# B&R Automation Studio project SMA_DATA
Automation Studio 4.8.7.28 SP

## Configuration PC

CPU PC_any, AutomationRuntime M4.93, Build 6.3.0, Vc V4.73.1

### Hardware
```
PC : PC_any v1.1.1.0 (OrderNumber=PC)
  ConfigurationID = SMA_DATA_PC
  Cyclic1Duration = 10000
  Cyclic1Tolerance = 100000
  FileDevice1
  FileDeviceName1 = USER
  FileDevicePath1 = USER_PATH
  ActivateOpcUa = 1
  OpcUaInformationModels_PV_Version = 1
```

## Configuration x1586

CPU X20CP1586, AutomationRuntime J4.93, Build 6.3.0, Vc V4.73.1

### Task classes (Cpu.sw)
```
Cyclic#1:
  DataSQL <- DataSQL.prg
  DataSQLPro <- DataSQLProduct.prg
Binaries: udbdef, FWRules, TCData, iomap, ashwac, Role, sysconf, arconfig, asfw, User, ashwd
Libraries: standard, AsBrStr
```

### Hardware
```
X20CP1586 : X20CP1586 v1.13.0.0
  Connector IF1:
    ActivateIna = 0
  Connector IF2:
    ActivateDevice = 1
    Mode = Manual
    InternetAddress = 192.168.50.233
    SubnetMask = 255.255.255.0
    InaPort = 11160
    ActivateSnmp = 2
  ConfigurationID = SMA_DATA_PC
  Simulation = 1
  Cyclic1Tolerance = 100000
  FileDevice1
  FileDeviceName1 = USER
  FileDevicePath1 = USER_PATH
  ActivateOpcUa = 1
  OpcUaInformationModels_PV_Version = 1
```

## Logical view

Binary libraries used (declarations not repeated): operator, runtime, astime, AsIecCon, standard, AsBrStr

### Package Logical/Libraries - Global libraries

### GlobalDataSQL.typ
```iecst
(*Global Data SQL Struct*)

TYPE
	DataSQLOperate_typ : 	STRUCT
		RecipeRead : BOOL;
		RecipeReadStatus : UINT;
		RecipeInsert : BOOL;
		RecipeInsertReq : BOOL;
		ProductRead : BOOL;
		ProductReadStatus : UINT;
		ProductInsert : BOOL;
		ProductInsertReq : BOOL;
		AuditRead : BOOL;
		AuditReadStatus : UINT;
		AuditInsertFault : BOOL;
		AlarmRead : BOOL;
		AlarmReadStatus : UINT;
		AlarmInsertFault : BOOL;
	END_STRUCT;
END_TYPE

(*Global Data SQL Struct*)

TYPE
	DataSQLQueryConfig_typ : 	STRUCT
		StartTime : ARRAY[0..READ_QUERY_SIZE_MINUS]OF STRING[20];
		EndTime : ARRAY[0..READ_QUERY_SIZE_MINUS]OF STRING[20];
		PointName : ARRAY[0..READ_QUERY_SIZE_MINUS]OF STRING[20];
		AuxQuery : ARRAY[0..READ_QUERY_SIZE_MINUS]OF STRING[80];
	END_STRUCT;
	DataSQLQueryCmd_typ : 	STRUCT
		Next : BOOL;
	END_STRUCT;
	DataSQLQuery_typ : 	STRUCT
		Config : DataSQLQueryConfig_typ;
		Cmd : DataSQLQueryCmd_typ;
	END_STRUCT;
END_TYPE

(*Global Data Struct - Recipe*)

TYPE
	DataSQLRecipe_typ : 	STRUCT
		TimeStamp : ARRAY[0..REV_BUFFER_SIZE_MINUS]OF DATE_AND_TIME;
		TimeStampTS : ARRAY[0..REV_BUFFER_SIZE_MINUS]OF UDINT;
		TimeStampFB : UDINT;
		State : ARRAY[0..REV_BUFFER_SIZE_MINUS]OF UDINT;
		StateTS : ARRAY[0..REV_BUFFER_SIZE_MINUS]OF UDINT;
		StateFB : UDINT;
		CH00 : ARRAY[0..REV_BUFFER_SIZE_MINUS]OF REAL;
		CH01 : ARRAY[0..REV_BUFFER_SIZE_MINUS]OF REAL;
		CH02 : ARRAY[0..REV_BUFFER_SIZE_MINUS]OF REAL;
		CH03 : ARRAY[0..REV_BUFFER_SIZE_MINUS]OF REAL;
		CH04 : ARRAY[0..REV_BUFFER_SIZE_MINUS]OF REAL;
		CH05 : ARRAY[0..REV_BUFFER_SIZE_MINUS]OF REAL;
		CH06 : ARRAY[0..REV_BUFFER_SIZE_MINUS]OF REAL;
		CH07 : ARRAY[0..REV_BUFFER_SIZE_MINUS]OF REAL;
		CH08 : ARRAY[0..REV_BUFFER_SIZE_MINUS]OF REAL;
		CH09 : ARRAY[0..REV_BUFFER_SIZE_MINUS]OF REAL;
		CH10 : ARRAY[0..REV_BUFFER_SIZE_MINUS]OF REAL;
		CH11 : ARRAY[0..REV_BUFFER_SIZE_MINUS]OF REAL;
		CH12 : ARRAY[0..REV_BUFFER_SIZE_MINUS]OF REAL;
		CH13 : ARRAY[0..REV_BUFFER_SIZE_MINUS]OF REAL;
		CH14 : ARRAY[0..REV_BUFFER_SIZE_MINUS]OF REAL;
		CH15 : ARRAY[0..REV_BUFFER_SIZE_MINUS]OF REAL;
		CH16 : ARRAY[0..REV_BUFFER_SIZE_MINUS]OF REAL;
		CH17 : ARRAY[0..REV_BUFFER_SIZE_MINUS]OF REAL;
		CH18 : ARRAY[0..REV_BUFFER_SIZE_MINUS]OF REAL;
		CH19 : ARRAY[0..REV_BUFFER_SIZE_MINUS]OF REAL;
		CH20 : ARRAY[0..REV_BUFFER_SIZE_MINUS]OF REAL;
		CH21 : ARRAY[0..REV_BUFFER_SIZE_MINUS]OF REAL;
		CH22 : ARRAY[0..REV_BUFFER_SIZE_MINUS]OF REAL;
		CH23 : ARRAY[0..REV_BUFFER_SIZE_MINUS]OF REAL;
		CH24 : ARRAY[0..REV_BUFFER_SIZE_MINUS]OF REAL;
		CH25 : ARRAY[0..REV_BUFFER_SIZE_MINUS]OF REAL;
		TS00 : ARRAY[0..REV_BUFFER_SIZE_MINUS]OF UDINT;
		TS01 : ARRAY[0..REV_BUFFER_SIZE_MINUS]OF UDINT;
		TS02 : ARRAY[0..REV_BUFFER_SIZE_MINUS]OF UDINT;
		TS03 : ARRAY[0..REV_BUFFER_SIZE_MINUS]OF UDINT;
		TS04 : ARRAY[0..REV_BUFFER_SIZE_MINUS]OF UDINT;
		TS05 : ARRAY[0..REV_BUFFER_SIZE_MINUS]OF UDINT;
		TS06 : ARRAY[0..REV_BUFFER_SIZE_MINUS]OF UDINT;
		TS07 : ARRAY[0..REV_BUFFER_SIZE_MINUS]OF UDINT;
		TS08 : ARRAY[0..REV_BUFFER_SIZE_MINUS]OF UDINT;
		TS09 : ARRAY[0..REV_BUFFER_SIZE_MINUS]OF UDINT;
		TS10 : ARRAY[0..REV_BUFFER_SIZE_MINUS]OF UDINT;
		TS11 : ARRAY[0..REV_BUFFER_SIZE_MINUS]OF UDINT;
		TS12 : ARRAY[0..REV_BUFFER_SIZE_MINUS]OF UDINT;
		TS13 : ARRAY[0..REV_BUFFER_SIZE_MINUS]OF UDINT;
		TS14 : ARRAY[0..REV_BUFFER_SIZE_MINUS]OF UDINT;
		TS15 : ARRAY[0..REV_BUFFER_SIZE_MINUS]OF UDINT;
		TS16 : ARRAY[0..REV_BUFFER_SIZE_MINUS]OF UDINT;
		TS17 : ARRAY[0..REV_BUFFER_SIZE_MINUS]OF UDINT;
		TS18 : ARRAY[0..REV_BUFFER_SIZE_MINUS]OF UDINT;
		TS19 : ARRAY[0..REV_BUFFER_SIZE_MINUS]OF UDINT;
		TS20 : ARRAY[0..REV_BUFFER_SIZE_MINUS]OF UDINT;
		TS21 : ARRAY[0..REV_BUFFER_SIZE_MINUS]OF UDINT;
		TS22 : ARRAY[0..REV_BUFFER_SIZE_MINUS]OF UDINT;
		TS23 : ARRAY[0..REV_BUFFER_SIZE_MINUS]OF UDINT;
		TS24 : ARRAY[0..REV_BUFFER_SIZE_MINUS]OF UDINT;
		TS25 : ARRAY[0..REV_BUFFER_SIZE_MINUS]OF UDINT;
		FB00 : UDINT;
		FB01 : UDINT;
		FB02 : UDINT;
		FB03 : UDINT;
		FB04 : UDINT;
		FB05 : UDINT;
		FB06 : UDINT;
		FB07 : UDINT;
		FB08 : UDINT;
		FB09 : UDINT;
		FB10 : UDINT;
		FB11 : UDINT;
		FB12 : UDINT;
		FB13 : UDINT;
		FB14 : UDINT;
		FB15 : UDINT;
		FB16 : UDINT;
		FB17 : UDINT;
		FB18 : UDINT;
		FB19 : UDINT;
		FB20 : UDINT;
		FB21 : UDINT;
		FB22 : UDINT;
		FB23 : UDINT;
		FB24 : UDINT;
		FB25 : UDINT;
	END_STRUCT;
END_TYPE

(*Global Data Struct - Product*)

TYPE
	DataSQLProduct_typ : 	STRUCT
		TimeStamp : ARRAY[0..REV_BUFFER_SIZE_MINUS]OF DATE_AND_TIME;
		TimeStampTS : ARRAY[0..REV_BUFFER_SIZE_MINUS]OF UDINT;
		TimeStampFB : UDINT;
		State : ARRAY[0..REV_BUFFER_SIZE_MINUS]OF UDINT;
		StateTS : ARRAY[0..REV_BUFFER_SIZE_MINUS]OF UDINT;
		StateFB : UDINT;
		CH01 : ARRAY[0..REV_BUFFER_SIZE_MINUS]OF REAL;
		CH02 : ARRAY[0..REV_BUFFER_SIZE_MINUS]OF REAL;
		CH03 : ARRAY[0..REV_BUFFER_SIZE_MINUS]OF REAL;
		CH04 : ARRAY[0..REV_BUFFER_SIZE_MINUS]OF REAL;
		CH05 : ARRAY[0..REV_BUFFER_SIZE_MINUS]OF REAL;
		CH06 : ARRAY[0..REV_BUFFER_SIZE_MINUS]OF REAL;
		TS01 : ARRAY[0..REV_BUFFER_SIZE_MINUS]OF UDINT;
		TS02 : ARRAY[0..REV_BUFFER_SIZE_MINUS]OF UDINT;
		TS03 : ARRAY[0..REV_BUFFER_SIZE_MINUS]OF UDINT;
		TS04 : ARRAY[0..REV_BUFFER_SIZE_MINUS]OF UDINT;
		TS05 : ARRAY[0..REV_BUFFER_SIZE_MINUS]OF UDINT;
		TS06 : ARRAY[0..REV_BUFFER_SIZE_MINUS]OF UDINT;
		FB01 : UDINT;
		FB02 : UDINT;
		FB03 : UDINT;
		FB04 : UDINT;
		FB05 : UDINT;
		FB06 : UDINT;
	END_STRUCT;
END_TYPE

(*Global Data Struct - Alarm*)

TYPE
	DataSQLAlarm_typ : 	STRUCT
		AlarmIndex : ARRAY[0..REV_BUFFER_SIZE_MINUS]OF UDINT;
		AlarmCode : ARRAY[0..REV_BUFFER_SIZE_MINUS]OF UDINT;
		AlarmCodeTS : ARRAY[0..REV_BUFFER_SIZE_MINUS]OF UDINT;
		AlarmCodeFB : ARRAY[0..REV_BUFFER_SIZE_MINUS]OF UDINT;
		AlarmTime : ARRAY[0..REV_BUFFER_SIZE_MINUS]OF DATE_AND_TIME;
		AlarmTimeTS : ARRAY[0..REV_BUFFER_SIZE_MINUS]OF UDINT;
		AlarmTimeFB : ARRAY[0..REV_BUFFER_SIZE_MINUS]OF UDINT;
		AlarmText : ARRAY[0..REV_BUFFER_SIZE_MINUS]OF WSTRING[50];
		AlarmTextTS : ARRAY[0..REV_BUFFER_SIZE_MINUS]OF UDINT;
		AlarmTextFB : ARRAY[0..REV_BUFFER_SIZE_MINUS]OF UDINT;
		AlarmState : ARRAY[0..REV_BUFFER_SIZE_MINUS]OF UDINT;
		AlarmStateTS : ARRAY[0..REV_BUFFER_SIZE_MINUS]OF UDINT;
		AlarmStateFB : ARRAY[0..REV_BUFFER_SIZE_MINUS]OF UDINT;
		AlarmStateStr : ARRAY[0..REV_BUFFER_SIZE_MINUS]OF STRING[80];
		AlarmLastItemIndex : UDINT;
	END_STRUCT;
END_TYPE

(*Global Data Struct - Audit*)

TYPE
	DataSQLAudit_typ : 	STRUCT
		AuditIndex : ARRAY[0..REV_BUFFER_SIZE_MINUS]OF UDINT;
		AuditTime : ARRAY[0..REV_BUFFER_SIZE_MINUS]OF DATE_AND_TIME;
		AuditTimeTS : ARRAY[0..REV_BUFFER_SIZE_MINUS]OF UDINT;
		AuditTimeFB : ARRAY[0..REV_BUFFER_SIZE_MINUS]OF UDINT;
		AuditOperator : ARRAY[0..REV_BUFFER_SIZE_MINUS]OF WSTRING[15];
		AuditOperatorTS : ARRAY[0..REV_BUFFER_SIZE_MINUS]OF UDINT;
		AuditOperatorFB : ARRAY[0..REV_BUFFER_SIZE_MINUS]OF UDINT;
		AuditText : ARRAY[0..REV_BUFFER_SIZE_MINUS]OF WSTRING[100];
		AuditTextTS : ARRAY[0..REV_BUFFER_SIZE_MINUS]OF UDINT;
		AuditTextFB : ARRAY[0..REV_BUFFER_SIZE_MINUS]OF UDINT;
		AuditTextReport : ARRAY[0..REV_BUFFER_SIZE_MINUS]OF WSTRING[100];
		AuditLastItemIndex : UDINT;
	END_STRUCT;
END_TYPE

(*Global Data Struct - Product*)

TYPE
	DataProduct_typ : 	STRUCT
		TimeStamp : DATE_AND_TIME;
		State : UDINT;
		CH01 : REAL;
		CH02 : REAL;
		CH03 : REAL;
		CH04 : REAL;
		CH05 : REAL;
		CH06 : REAL;
	END_STRUCT;
END_TYPE
```

### GlobalDataSQL.var
```iecst
(*Global DataSQL Constant*)
VAR CONSTANT
	REV_BUFFER_SIZE : UINT := 2000;
	REV_BUFFER_SIZE_MINUS : UINT := REV_BUFFER_SIZE-1;
	READ_QUERY_SIZE : UINT := 30;
	READ_QUERY_SIZE_MINUS : UINT := READ_QUERY_SIZE-1;
	READ_QUERY_SIZE_RCP : UINT := 27;
	READ_QUERY_SIZE_RCP_MINUS : UINT := READ_QUERY_SIZE_RCP-1;
	READ_QUERY_SIZE_PRO : UINT := 8;
	READ_QUERY_SIZE_PRO_MINUS : UINT := READ_QUERY_SIZE_PRO-1;
	READ_QUERY_SIZE_ALARM : UINT := 4;
	READ_QUERY_SIZE_ALARM_MINUS : UINT := READ_QUERY_SIZE_ALARM-1;
	READ_QUERY_SIZE_AUDIT : UINT := 3;
	READ_QUERY_SIZE_AUDIT_MINUS : UINT := READ_QUERY_SIZE_AUDIT-1;
END_VAR
(*Global DataSQL Constant*)
VAR CONSTANT
	DATA_ALARM_NUM : USINT := 100;
	DATA_ALARM_NUM_MINUS : USINT := DATA_ALARM_NUM-1;
	DATA_AUDIT_NUM : USINT := 100;
	DATA_AUDIT_NUM_MINUS : USINT := DATA_AUDIT_NUM-1;
	QUERY_TIME_OFFSET : DATE_AND_TIME := DT#1970-01-01-00:05:00;
END_VAR
(*Global DataSQL Variable*)
VAR
	gDataSQLHeartBeat : UINT;
	gDataSQLCommFault : BOOL;
	gDataSQLOperate : DataSQLOperate_typ;
	gDataSQLProduct : DataProduct_typ;
END_VAR
```

### Program Logical/DataSQL (ANSIC)

#### DataSQL.c - Init, cyclic, exit code
```c
#include <bur/plctypes.h>

#ifdef _DEFAULT_INCLUDES
	#include <AsDefault.h>
#endif

void _INIT DataSQLInit(void)
{
	gDataSQLHeartBeat = 0;
}

void _CYCLIC DataSQLCyclic(void)
{
	//通讯状态检测
	TimerDataSQLComm.IN = !gDataSQLHeartBeat;
	TimerDataSQLComm.PT = 1000;
	TON_10ms(&TimerDataSQLComm);

	if(TimerDataSQLComm.Q)
	{
		gDataSQLCommFault = 1;
	}

	if(gDataSQLHeartBeat==1)
	{
		gDataSQLHeartBeat = 0;
	}
}

void _EXIT DataSQLExit(void)
{

}
```

#### DataSQL.var - Local variables
```iecst
(*Data SQL Variable*)
VAR
	TimerDataSQLComm : TON_10ms;
END_VAR
```

### Program Logical/DataSQLProduct (ANSIC)

#### DataSQLProduct.c - Init, cyclic, exit code
```c
#include <bur/plctypes.h>

#ifdef _DEFAULT_INCLUDES
	#include <AsDefault.h>
#endif

void _INIT DataSQLProductInit(void)
{
	ProductDataSQLRev.FB01 = 0;

	for(int i=0; i<READ_QUERY_SIZE; i++)
	{
		brsstrcpy(ProductDataSQLQuery.Config.StartTime[i], "2026-4-1 10:00:00");
		brsstrcpy(ProductDataSQLQuery.Config.EndTime[i],   "2026-6-1 10:00:00");
	}
}

void _CYCLIC DataSQLProductCyclic(void)
{
	/*******************************************************生产数据查询*******************************************************/
	//系统功能 - 当前系统时间
	SystemGetTime.enable = 1;
	DTGetTime(&SystemGetTime);

	SystemTimeAct = SystemGetTime.DT1;

	//生产数据存储
	if(gDataSQLOperate.ProductInsertReq)
	{
		gDataSQLOperate.ProductInsertReq = 0;
		gDataSQLOperate.ProductInsert	 = 1;

		//生产数据锁存
		gDataSQLProduct.TimeStamp = SystemTimeAct;
		gDataSQLProduct.State  	  = 2;
		gDataSQLProduct.CH01	  = 1;
		gDataSQLProduct.CH02	  = 2;
		gDataSQLProduct.CH03	  = 3;
		gDataSQLProduct.CH04	  = 4;
		gDataSQLProduct.CH05	  = 5;
		gDataSQLProduct.CH06	  = 6;
	}

	/*******************************************************生产数据查询*******************************************************/
	//生产数据查询配置
	brsstrcpy(ProductDataSQLQuery.Config.PointName[0], "DataProductTime");
	brsstrcpy(ProductDataSQLQuery.Config.PointName[1], "DataProductState");
	brsstrcpy(ProductDataSQLQuery.Config.PointName[2], "DataProductCH01");
	brsstrcpy(ProductDataSQLQuery.Config.PointName[3], "DataProductCH02");
	brsstrcpy(ProductDataSQLQuery.Config.PointName[4], "DataProductCH03");
	brsstrcpy(ProductDataSQLQuery.Config.PointName[5], "DataProductCH04");
	brsstrcpy(ProductDataSQLQuery.Config.PointName[6], "DataProductCH05");
	brsstrcpy(ProductDataSQLQuery.Config.PointName[7], "DataProductCH06");

	//生产数据查询缓存
	ProductDataSQLRev;
}

void _EXIT DataSQLProductExit(void)
{

}
```

#### DataSQLProduct.var - Local variables
```iecst
(*Data SQL Variable - Product*)
VAR
	ProductDataSQLQuery : DataSQLQuery_typ;
	ProductDataSQLRev : DataSQLProduct_typ;
	SystemGetTime : DTGetTime;
	SystemTimeAct : DATE_AND_TIME;
END_VAR
```

Listed in the project but not available here: Logical/Global.typ, Logical/Global.var, Logical/DataSQL/DataSQL.typ, Logical/DataSQLProduct/DataSQLProduct.typ
